// TIA Portal V16 export
// export: Created 2022-11-17T11:55:32.5696507Z, ExportSetting WithDefaults, DisplayName Totally Integrated Automation Portal, DisplayVersion V16 Update 6, DisplayName TIA Portal Version Control Interface, DisplayVersion V16 Update 2, DisplayName TIA Portal Openness, DisplayVersion V16 Update 6, DisplayName SINAMICS Startdrive Advanced, DisplayVersion V16 Update 5, DisplayName SINAMICS Startdrive G130, G150, S120, S150, SINAMICS MV, S210, DisplayVersion V16 Update 5, DisplayName SINAMICS Startdrive G110M, G120, G120C, G120D, G120P, G115D, DisplayVersion V16 Update 5, DisplayName STEP 7 Professional, DisplayVersion V16 Update 6, DisplayName STEP 7 Safety, DisplayVersion V16, DisplayName WinCC Advanced, DisplayVersion V16 Update 6
DATA_BLOCK "DB236_Program14"   // DB236
{ S7_Optimized_Access := 'FALSE' }
AUTHOR : Robopac
VERSION : 0.0
// stored: AutoNumber false, IsOnlyStoredInLoadMemory false, IsWriteProtectedInAS false
   VAR RETAIN
      Program14 { S7_SetPoint := 'True'} : "DatiProgramma";
   END_VAR
BEGIN
   Program14.Wrapping := TRUE;
   Program14.TopLenght := 500;
   Program14.TopRelease := 0;
   Program14.TopDown := 0;
   Program14.Top := 4;
   Program14.PressurePTime := 0;
   Program14.LifterTime := 0;
   Program14.RevOverContrast := 1;
   Program14.RopeEndCycle := 16#02;
   Program14.Spare4 := 16#01;
   Program14.RopeTime := 1500;
   Program14.RevOverClamp := 1;
   Program14.FilmForceFinalRev := 10;
   Program14.FilmPrestretchFinalRev := 100;
   Program14.ArmSpeed := 100;
   Program14.CarriageDown4Top := 500;
   Program14.TopDownTime := 1500;
   Program14.LapsUnderTop := 0;
   Program14.Spare6 := 0;
   Program14.Spare7 := 0;
   Program14.Spare8 := 0;
   Program14.Spare9 := 0;
   Program14.Spare10 := 0;
   Program14.Spare11 := 0;
   Program14.Spare12 := 0;
   Program14.Overlap0_1 := 0;
   Program14.Height1 := 130;
   Program14.Landmark1 := FALSE;
   Program14.Lifter1 := FALSE;
   Program14.SpareBit1H1 := FALSE;
   Program14.Airblower1 := TRUE;
   Program14.NextStep1 := TRUE;
   Program14.PressureP1 := TRUE;
   Program14.SpareByte2H1 := 16#00;
   Program14.Revolution1 := 1;
   Program14.RopeUnit1_1 := 16#01;
   Program14.RopeUnit1_2 := 16#01;
   Program14.FilmForce1 := 5;
   Program14.FilmPrestretch1 := 200;
   Program14.Spare3H1 := 0;
   Program14.Spare49 := 0;
   Program14.Spare50 := 0;
   Program14.Spare51 := 0;
   Program14.Spare52 := 0;
   Program14.Spare53 := 0;
   Program14.Overlap1_2 := 0;
   Program14.Height2 := 50;
   Program14.Landmark2 := FALSE;
   Program14.Lifter2 := FALSE;
   Program14.SpareBit1H2 := FALSE;
   Program14.Airblower2 := TRUE;
   Program14.NextStep2 := TRUE;
   Program14.PressureP2 := TRUE;
   Program14.SpareByte2H2 := 16#00;
   Program14.Revolution2 := 1;
   Program14.RopeUnit2_1 := 16#01;
   Program14.RopeUnit2_2 := 16#01;
   Program14.FilmForce2 := 20;
   Program14.FilmPrestretch2 := 200;
   Program14.Spare3H2 := 0;
   Program14.Spare54 := 0;
   Program14.Spare55 := 0;
   Program14.Spare56 := 0;
   Program14.Spare57 := 0;
   Program14.Spare58 := 0;
   Program14.Overlap2_3 := 100;
   Program14.Height3 := -50;
   Program14.Landmark3 := TRUE;
   Program14.Lifter3 := FALSE;
   Program14.SpareBit1H3 := FALSE;
   Program14.Airblower3 := TRUE;
   Program14.NextStep3 := TRUE;
   Program14.PressureP3 := TRUE;
   Program14.SpareByte2H3 := 16#00;
   Program14.Revolution3 := 2;
   Program14.RopeUnit3_1 := 16#01;
   Program14.RopeUnit3_2 := 16#01;
   Program14.FilmForce3 := 30;
   Program14.FilmPrestretch3 := 200;
   Program14.Spare3H3 := 0;
   Program14.Spare59 := 0;
   Program14.Spare60 := 0;
   Program14.Spare61 := 380;
   Program14.Spare62 := 2800;
   Program14.Spare63 := 0;
   Program14.Overlap3_4 := 100;
   Program14.Height4 := 100;
   Program14.Landmark4 := FALSE;
   Program14.Lifter4 := FALSE;
   Program14.SpareBit1H4 := FALSE;
   Program14.Airblower4 := TRUE;
   Program14.NextStep4 := TRUE;
   Program14.PressureP4 := TRUE;
   Program14.SpareByte2H4 := 16#00;
   Program14.Revolution4 := 3;
   Program14.RopeUnit4_1 := 16#02;
   Program14.RopeUnit4_2 := 16#02;
   Program14.FilmForce4 := 30;
   Program14.FilmPrestretch4 := 200;
   Program14.Spare3H4 := 0;
   Program14.Spare64 := 0;
   Program14.Spare65 := 0;
   Program14.Spare66 := 0;
   Program14.Spare67 := 0;
   Program14.Spare68 := 0;
   Program14.Overlap4_5 := 0;
   Program14.Height5 := 50;
   Program14.Landmark5 := FALSE;
   Program14.Lifter5 := FALSE;
   Program14.SpareBit1H5 := FALSE;
   Program14.Airblower5 := TRUE;
   Program14.NextStep5 := FALSE;
   Program14.PressureP5 := FALSE;
   Program14.SpareByte2H5 := 16#00;
   Program14.Revolution5 := 1;
   Program14.RopeUnit5_1 := 16#01;
   Program14.RopeUnit5_2 := 16#01;
   Program14.FilmForce5 := 30;
   Program14.FilmPrestretch5 := 200;
   Program14.Spare3H5 := 0;
   Program14.Spare69 := 0;
   Program14.Spare70 := 0;
   Program14.Spare71 := 0;
   Program14.Spare72 := 0;
   Program14.Spare73 := 0;
   Program14.Overlap5_6 := 100;
   Program14.Height6 := 50;
   Program14.Landmark6 := FALSE;
   Program14.Lifter6 := FALSE;
   Program14.SpareBit1H6 := FALSE;
   Program14.Airblower6 := TRUE;
   Program14.NextStep6 := FALSE;
   Program14.PressureP6 := FALSE;
   Program14.SpareByte2H6 := 16#00;
   Program14.Revolution6 := 2;
   Program14.RopeUnit6_1 := 16#02;
   Program14.RopeUnit6_2 := 16#01;
   Program14.FilmForce6 := 20;
   Program14.FilmPrestretch6 := 200;
   Program14.Spare3H6 := 0;
   Program14.Spare74 := 0;
   Program14.Spare75 := 0;
   Program14.Spare76 := 0;
   Program14.Spare77 := 0;
   Program14.Spare78 := 0;
   Program14.Overlap6_7 := 0;
   Program14.Height7 := 0;
   Program14.Landmark7 := FALSE;
   Program14.Lifter7 := FALSE;
   Program14.SpareBit1H7 := FALSE;
   Program14.Airblower7 := FALSE;
   Program14.NextStep7 := TRUE;
   Program14.PressureP7 := FALSE;
   Program14.SpareByte2H7 := 16#00;
   Program14.Revolution7 := 1;
   Program14.RopeUnit7_1 := 16#01;
   Program14.RopeUnit7_2 := 16#01;
   Program14.FilmForce7 := 0;
   Program14.FilmPrestretch7 := 100;
   Program14.Spare3H7 := 0;
   Program14.Spare79 := 0;
   Program14.Spare80 := 0;
   Program14.Spare81 := 0;
   Program14.Spare82 := 0;
   Program14.Spare83 := 0;
   Program14.Overlap7_8 := 0;
   Program14.Height8 := 0;
   Program14.Landmark8 := FALSE;
   Program14.Lifter8 := FALSE;
   Program14.SpareBit1H8 := FALSE;
   Program14.Airblower8 := FALSE;
   Program14.NextStep8 := TRUE;
   Program14.PressureP8 := FALSE;
   Program14.SpareByte2H8 := 16#00;
   Program14.Revolution8 := 1;
   Program14.RopeUnit8_1 := 16#01;
   Program14.RopeUnit8_2 := 16#01;
   Program14.FilmForce8 := 0;
   Program14.FilmPrestretch8 := 100;
   Program14.Spare3H8 := 0;
   Program14.Spare84 := 0;
   Program14.Spare85 := 0;
   Program14.Spare86 := 0;
   Program14.Spare87 := 0;
   Program14.Spare88 := 0;
   Program14.Overlap8_9 := 0;
   Program14.Height9 := 0;
   Program14.Landmark9 := FALSE;
   Program14.Lifter9 := FALSE;
   Program14.SpareBit1H9 := FALSE;
   Program14.Airblower9 := FALSE;
   Program14.NextStep9 := TRUE;
   Program14.PressureP9 := FALSE;
   Program14.SpareByte2H9 := 16#00;
   Program14.Revolution9 := 1;
   Program14.RopeUnit9_1 := 16#01;
   Program14.RopeUnit9_2 := 16#01;
   Program14.FilmForce9 := 0;
   Program14.FilmPrestretch9 := 100;
   Program14.Spare3H9 := 0;
   Program14.Spare89 := 0;
   Program14.Spare90 := 0;
   Program14.Spare91 := 0;
   Program14.Spare92 := 0;
   Program14.Spare93 := 0;
   Program14.Overlap9_10 := 0;
   Program14.Height10 := 0;
   Program14.Landmark10 := FALSE;
   Program14.Lifter10 := FALSE;
   Program14.SpareBit1H10 := FALSE;
   Program14.Airblower10 := FALSE;
   Program14.NextStep10 := FALSE;
   Program14.PressureP10 := FALSE;
   Program14.SpareByte2H10 := 16#00;
   Program14.Revolution10 := 1;
   Program14.RopeUnit10_1 := 16#01;
   Program14.RopeUnit10_2 := 16#01;
   Program14.FilmForce10 := 0;
   Program14.FilmPrestretch10 := 100;
   Program14.Spare3H10 := 0;
   Program14.Spare94 := 0;
   Program14.Spare95 := 0;
   Program14.Spare96 := 0;
   Program14.Spare97 := 0;
   Program14.Spare98 := 0;
   Program14.Overlap10_11 := 0;
   Program14.Height11 := 0;
   Program14.Landmark11 := FALSE;
   Program14.Lifter11 := FALSE;
   Program14.SpareBit1H11 := FALSE;
   Program14.Airblower11 := FALSE;
   Program14.NextStep11 := TRUE;
   Program14.PressureP11 := FALSE;
   Program14.SpareByte2H11 := 16#00;
   Program14.Revolution11 := 1;
   Program14.RopeUnit11_1 := 16#01;
   Program14.RopeUnit11_2 := 16#01;
   Program14.FilmForce11 := 0;
   Program14.FilmPrestretch11 := 100;
   Program14.Spare3H11 := 0;
   Program14.Spare99 := 0;
   Program14.Spare100 := 0;
   Program14.Spare101 := 0;
   Program14.Spare102 := 0;
   Program14.Spare103 := 0;
   Program14.Overlap11_12 := 0;
   Program14.Height12 := 0;
   Program14.Landmark12 := FALSE;
   Program14.Lifter12 := FALSE;
   Program14.SpareBit1H12 := FALSE;
   Program14.Airblower12 := FALSE;
   Program14.NextStep12 := FALSE;
   Program14.PressureP12 := FALSE;
   Program14.SpareByte2H12 := 16#00;
   Program14.Revolution12 := 1;
   Program14.RopeUnit12_1 := 16#01;
   Program14.RopeUnit12_2 := 16#01;
   Program14.FilmForce12 := 0;
   Program14.FilmPrestretch12 := 100;
   Program14.Spare3H12 := 0;
   Program14.Spare104 := 0;
   Program14.Spare105 := 0;
   Program14.Spare106 := 0;
   Program14.Spare107 := 0;
   Program14.Spare108 := 0;
END_DATA_BLOCK
